{attribute 'qualified_only'}
VAR_GLOBAL
	M_Group1ClampOpen :BOOL;
	M_Group2ClampOpen :BOOL;
	M_TT_0 : BOOL;
	M_Trunion_0 : BOOL;
	M_Door_Cls : BOOL;
	M_HomeDone : Bool;
END_VAR

(* stored: Version 1.1.0.1, ProductVersion 3.1.4024.16
   GVL Home_Seq_DB: Id {19cc2f80-a007-4d5d-b787-b04a9682f174} *)
